(* CODESYS project 02_demo.project

Project tree, tasks and I/O mapping:
  Device : CODESYS Control arm CTH3 C37-001S2v28, 3S - Smart Software Solutions GmbH, version 3.5.4.30
    application Application
      libraries: Standard, * (System)
      task MainTask (cyclic, interval t#20ms, priority 1) calls PLC_PRG
      task EtherCAT_Master (cyclic, interval 4000 µs, priority 0) calls EtherCAT_Master.EtherCAT_Task [EtherCAT_Master.EtherCAT_Task], POU
      program PLC_PRG [ST]
      program POU [ST]
    SoftMotion General Axis Pool
    Co-trust LocalBus
    EtherCAT_Master : EtherCAT Master, 3S - Smart Software Solutions GmbH, version 3.5.4.0
        settings: NetworkName = 'eth3'; SelectNetworkByName = True
      A4N_EtherCAT : A4N EtherCAT V2.00, COTRUST, version Revision=16#00000002
          settings: EnableExpertSettings = True; DC sync0 cycletime = 4000; DC sync1 cycletime = 4000
          unmapped channels: Controlword, target position, target torque, max profile velocity, target velocity, touch probe function, Mode of operation, Statusword, position actual value, velocity actual value, torque actual value, mode of operation display, Touch probe status, touch probe pos1 pos value, touch probe pos1 neg value, Digital input
        dbgAxis : SM_Drive_GenericDSP402, 3S - Smart Software Solutions GmbH, order no. 0, version 3.5.4.10
            settings: bVirtual = TRUE; iMovementType = 0; fSWLimitDeceleration = 0.0; fSWErrorMaxDistance = 0.0; AdrOffset_8010 = 0; BitOffset_8010 = 0; BitLength_8010 = 16; Address_8010 = '%QW0'; Type_8010 = 'UINT'; AddressPointer_8010 = ADR(%QW0); AdrOffset_8020 = 4; BitOffset_8020 = 0; BitLength_8020 = 32; Address_8020 = '%QD1'; Type_8020 = 'DINT'; AddressPointer_8020 = ADR(%QD1); AdrOffset_8030 = 16; BitOffset_8030 = 0; BitLength_8030 = 32; Address_8030 = '%QD4'; Type_8030 = 'DINT'; AddressPointer_8030 = ADR(%QD4); AdrOffset_8040 = 8; BitOffset_8040 = 0; BitLength_8040 = 16; Address_8040 = '%QW4'; Type_8040 = 'INT'; AddressPointer_8040 = ADR(%QW4); AdrOffset_8050 = 22; BitOffset_8050 = 0; BitLength_8050 = 16; Address_8050 = '%QW11'; Type_8050 = 'INT'; AddressPointer_8050 = ADR(%QW11); AdrOffset_8060 = 20; BitOffset_8060 = 0; BitLength_8060 = 16; Address_8060 = '%QW10'; Type_8060 = 'UINT'; AddressPointer_8060 = ADR(%QW10);
              AdrOffset_8070 = 16#FFFFFFFF; BitOffset_8070 = 0; BitLength_8070 = 0; Address_8070 = ''; Type_8070 = ''; AddressPointer_8070 = 0; AdrOffset_8080 = 16#FFFFFFFF; BitOffset_8080 = 0; BitLength_8080 = 0; Address_8080 = ''; Type_8080 = ''; AddressPointer_8080 = 0; AdrOffset_8510 = 0; BitOffset_8510 = 0; BitLength_8510 = 16; Address_8510 = '%IW0'; Type_8510 = 'UINT'; AddressPointer_8510 = ADR(%IW0); AdrOffset_8520 = 4; BitOffset_8520 = 0; BitLength_8520 = 32; Address_8520 = '%ID1'; Type_8520 = 'DINT'; AddressPointer_8520 = ADR(%ID1); AdrOffset_8530 = 8; BitOffset_8530 = 0; BitLength_8530 = 32; Address_8530 = '%ID2'; Type_8530 = 'DINT'; AddressPointer_8530 = ADR(%ID2); AdrOffset_8540 = 12; BitOffset_8540 = 0; BitLength_8540 = 16; Address_8540 = '%IW6'; Type_8540 = 'INT'; AddressPointer_8540 = ADR(%IW6); AdrOffset_8550 = 14; BitOffset_8550 = 0; BitLength_8550 = 16; Address_8550 = '%IW7';
              Type_8550 = 'INT'; AddressPointer_8550 = ADR(%IW7); AdrOffset_8560 = 28; BitOffset_8560 = 0; BitLength_8560 = 32; Address_8560 = '%ID7'; Type_8560 = 'UDINT'; AddressPointer_8560 = ADR(%ID7); AdrOffset_8570 = 16; BitOffset_8570 = 0; BitLength_8570 = 16; Address_8570 = '%IW8'; Type_8570 = 'UINT'; AddressPointer_8570 = ADR(%IW8); AdrOffset_8580 = 20; BitOffset_8580 = 0; BitLength_8580 = 32; Address_8580 = '%ID5'; Type_8580 = 'DINT'; AddressPointer_8580 = ADR(%ID5); AdrOffset_8590 = 24; BitOffset_8590 = 0; BitLength_8590 = 32; Address_8590 = '%ID6'; Type_8590 = 'DINT'; AddressPointer_8590 = ADR(%ID6); AdrOffset_8600 = 16#FFFFFFFF; BitOffset_8600 = 0; BitLength_8600 = 0; Address_8600 = ''; Type_8600 = ''; AddressPointer_8600 = 0; AdrOffset_8600 = 16#FFFFFFFF; BitOffset_8600 = 0; BitLength_8600 = 0; Address_8610 = ''; Type_8610 = ''; AddressPointer_8610 = 0
*)

// Device/Application/PLC_PRG
PROGRAM PLC_PRG
VAR

END_VAR

END_PROGRAM

// Device/Application/POU
PROGRAM POU
VAR
	mcp: MC_Power; //使能函数
	mcmv: MC_Jog;  //点动函数
	mcmabs: MC_MoveAbsolute;	// 绝对值定位运动
	mcminc: MC_MoveRelative;	// 增量式运动
	MVStop: MC_Stop;			// 电机停止
	dbgAxisHome: MC_Home;			// 电机回零
	dbgAxisReset: MC_Reset;		// 电机故障复位
	Motionstate: INT := 1;			// 测试用，控制测试功能
	Cnt:INT;					// 仅仅用于测试

	Jog_Pos: BOOL ;				// 点动正 使能
	Jog_Neg: BOOL;				// 点动负 使能
	
	MovEnable: BOOL;			// 定位运行、回零及停止时的函数模块使能
	MovIncDistance: LREAL;		// 增量运动距离设定
	MV_Speed: LREAL;			// 运行速度设定
	MV_Acc: LREAL;				// 运行加速度设定
	MV_Dec: LREAL;				// 运行减速度设定
	MV_Jerk: LREAL;				// 运行加加速度设定
	
	MovAbsDistance: LREAL;		// 绝对定位时的目标位置
END_VAR


CASE Motionstate OF
0:
	Cnt := Cnt+1;
	MV_Speed:= 10000;
	MV_Acc:= 1000000;
	MV_Dec:= 1000000;
	MV_Jerk:= 100000000;
	Jog_Pos:= TRUE;
1: //Enable motor,Power on
mcp(
    Axis:= dbgAxis , 
    Enable:= TRUE , 
	bRegulatorOn:= TRUE,
	bDriveStart:= TRUE,
    Status=> , 
    Busy=> , 
    Error=> , 
    ErrorID=> );

2:// Disable motor,Power off
mcp(
    Axis:=dbgAxis , 
    Enable:= TRUE , 
	bRegulatorOn:= FALSE,
	bDriveStart:= TRUE,
    Status=> , 
    Busy=> , 
    Error=> , 
    ErrorID=> );

3: // JOG+ and JOG-
mcmv(
    Axis:=dbgAxis , 
    JogForward:=Jog_Pos , 
    JogBackward:=Jog_Neg , 

    Velocity:= MV_Speed, 
    Acceleration:= MV_Acc, 
    Deceleration:= MV_Dec, 
    Jerk:= MV_Jerk, 
    Busy=> , 
    CommandAborted=> , 
    Error=> , 
    ErrorID=> );

4: // Move relative POS and Neg
mcminc(
    Axis:=dbgAxis , 
	Execute:= MovEnable,
	Distance:= MovIncDistance,
    Velocity:= MV_Speed, 
    Acceleration:= MV_Acc, 
    Deceleration:= MV_Dec, 
    Jerk:= MV_Jerk, 
	Done=> ,
    Busy=> , 
    CommandAborted=> , 
    Error=> , 
    ErrorID=> );

5: // Move Abs
mcmabs(
    Axis:=dbgAxis , 
	Execute:= MovEnable,
	Position:= MovAbsDistance,
    Velocity:= MV_Speed, 
    Acceleration:= MV_Acc, 
    Deceleration:= MV_Dec, 
    Jerk:= MV_Jerk, 
	Done=> ,
    Busy=> , 
    CommandAborted=> , 
    Error=> , 
    ErrorID=> );


6: // Stop motor
MVStop(
    Axis:=dbgAxis , 
	Execute:= MovEnable,
    Jerk:= MV_Jerk, 
	Done=> ,
    Busy=> , 
    Error=> , 
    ErrorID=> );

	
7: // Home
dbgAxisHome(
    Axis:=dbgAxis , 
	Execute:= MovEnable,

	Done=> ,
    Busy=> , 
	CommandAborted=> , 
    Error=> , 
    ErrorID=> );
8:
dbgAxisReset(
    Axis:=dbgAxis , 
	Execute:= TRUE,
);	

END_CASE;

END_PROGRAM
